PROGRAM MAIN
VAR
END_VAR

GarageDoor();

END_PROGRAM

(* stored: Version 1.1.0.1, ProductVersion 3.1.4024.12
   POU MAIN: Id {cdad2e52-bd24-442a-ba65-805229cea4a5}, SpecialFunc None *)
